(* Logix 5000 project; controller Reto1_SCADA Emulate 5570 rev 30.12; software revision 30.00 *)

TASK MainTask (continuous, watchdog 500 ms) : MainProgram

MODULES
   Local : Emulate 5570 (ICP 2, rev 30.12)
      I_O : vendor 1 type 0 code 15 (ICP 3, rev 1.1, Output RPI 150 ms)
END_MODULES

VAR_GLOBAL   (* controller tags *)
   Ambas : BOOL;
   Avanza_Exit : BOOL;
   BandaCorrecta : BOOL := 1;
   Bandera : BOOL := 1;
   BanderaA : BOOL;
   BanderaAmbas : BOOL;
   BanderaV : BOOL;
   BanExitA : BOOL;
   BanExiV : BOOL;
   BanSenA : BOOL;
   BanSenV : BOOL;
   ContadorA : COUNTER := (ACC := 10);
   ContadorV : COUNTER := (ACC := 10);
   Detener_Exit : BOOL;
   FIO_Avanzar : BOOL;
   FIO_AvanzarA : BOOL := 1;
   FIO_AvanzarUPA : BOOL := 1;
   FIO_AvanzarUPV : BOOL := 1;
   FIO_AvanzarV : BOOL := 1;
   FIO_Banda1 : BOOL := 1;
   FIO_Banda1b : BOOL := 1;
   FIO_Banda2 : BOOL := 1;
   FIO_Banda2b : BOOL := 1;
   FIO_BanderaBanda : BOOL;
   FIO_BanderaBandaA : BOOL;
   FIO_BanderaBandaV : BOOL;
   FIO_Detener : BOOL;
   FIO_DetenerA : BOOL;
   FIO_DetenerV : BOOL;
   FIO_Iniciar : BOOL;
   FIO_IniciarA : BOOL;
   FIO_IniciarV : BOOL;
   FIO_ParadaUPA : BOOL;
   FIO_ParadaUPV : BOOL;
   FIO_PusherAzul : BOOL;
   FIO_PusherVerde : BOOL;
   FIO_SensorAzul : BOOL;
   FIO_SensorExitA : BOOL;
   FIO_SensorExitV : BOOL;
   FIO_SensorPaso1 : BOOL;
   FIO_SensorPaso2 : BOOL;
   FIO_SensorVerde : BOOL;
   FIO_Start : BOOL;
   FIO_Stop : BOOL := 1;
   FIO_Stop_emergencia : BOOL := 1;
   FlancoBajadaA : BOOL;
   FlancoBajadaExA : BOOL;
   FlancoBajadaExV : BOOL;
   FlancoBajadaV : BOOL;
   TimerAvan : TIMER := (PRE := 1000, ACC := 25, EN := 1, TT := 1);
   TimerAvanV : TIMER := (PRE := 1000, ACC := 22, EN := 1, TT := 1);
   TimerBanda : TIMER := (PRE := 3000);
   TimerBandaV : TIMER := (PRE := 3000);
   TimerBien : TIMER := (PRE := 500, ACC := 510, EN := 1, DN := 1);
   TimerInicio : TIMER := (PRE := 2000, ACC := 2022, EN := 1, DN := 1);
   TimerInicioV : TIMER := (PRE := 2000, ACC := 2015, EN := 1, DN := 1);
   TimerP : TIMER := (PRE := 4000);
   TimerPUN : TIMER := (PRE := 3000, ACC := 2020, TT := 1, DN := 1);
   TimerPUNV : TIMER := (PRE := 3000, ACC := 2015, TT := 1, DN := 1);
   TimerPV : TIMER := (PRE := 4000);
   TimerStart : TIMER := (PRE := 4000);
END_VAR

PROGRAM MainProgram   (* main routine MainRoutine *)

ROUTINE Azul   (* ladder *)
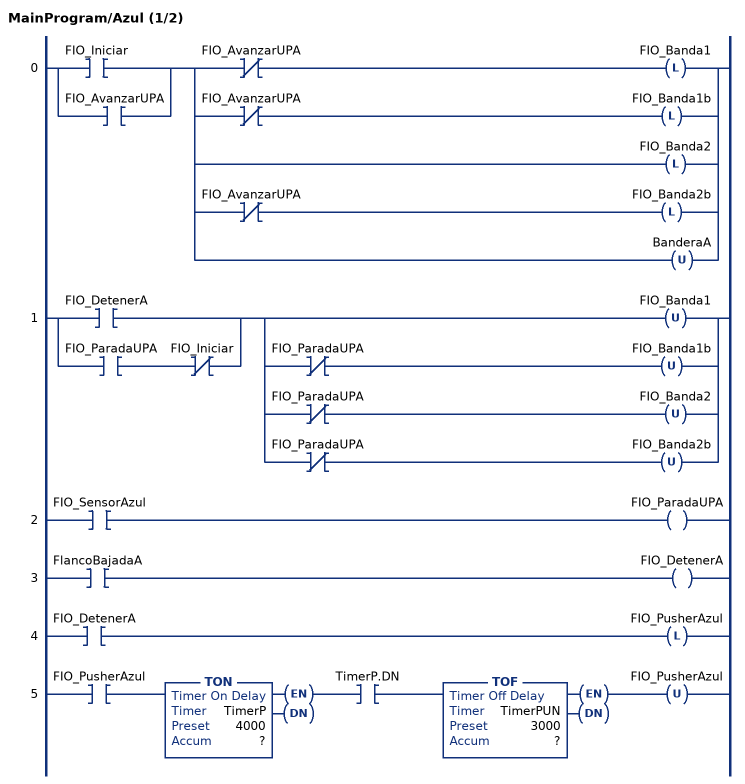
   0: [XIC(FIO_Iniciar) ,XIC(FIO_AvanzarUPA) ][XIO(FIO_AvanzarUPA) OTL(FIO_Banda1) ,XIO(FIO_AvanzarUPA) OTL(FIO_Banda1b) ,OTL(FIO_Banda2) ,XIO(FIO_AvanzarUPA) OTL(FIO_Banda2b) ,OTU(BanderaA) ];
   1: [XIC(FIO_DetenerA) ,XIC(FIO_ParadaUPA) XIO(FIO_Iniciar) ][OTU(FIO_Banda1) ,XIO(FIO_ParadaUPA) OTU(FIO_Banda1b) ,XIO(FIO_ParadaUPA) OTU(FIO_Banda2) ,XIO(FIO_ParadaUPA) OTU(FIO_Banda2b) ];
   2: XIC(FIO_SensorAzul)OTE(FIO_ParadaUPA);
   3: XIC(FlancoBajadaA)OTE(FIO_DetenerA);
   4: XIC(FIO_DetenerA)OTL(FIO_PusherAzul);
   5: XIC(FIO_PusherAzul)TON(TimerP,?,?)XIC(TimerP.DN)TOF(TimerPUN,?,?)OTU(FIO_PusherAzul);
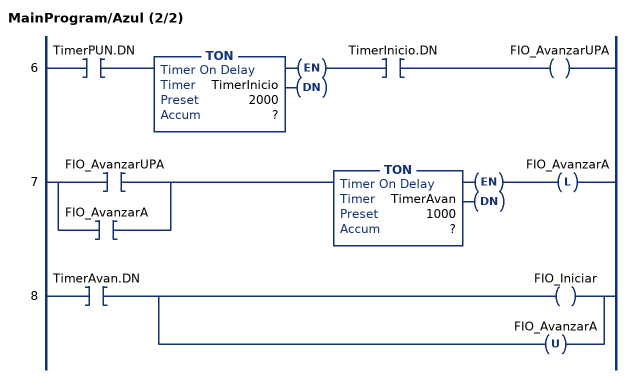
   6: XIC(TimerPUN.DN)TON(TimerInicio,?,?)XIC(TimerInicio.DN)OTE(FIO_AvanzarUPA);
   7: [XIC(FIO_AvanzarUPA) ,XIC(FIO_AvanzarA) ]TON(TimerAvan,?,?)OTL(FIO_AvanzarA);
   8: XIC(TimerAvan.DN)[OTE(FIO_Iniciar) ,OTU(FIO_AvanzarA) ];
END_ROUTINE

ROUTINE MainRoutine   (* ladder *)
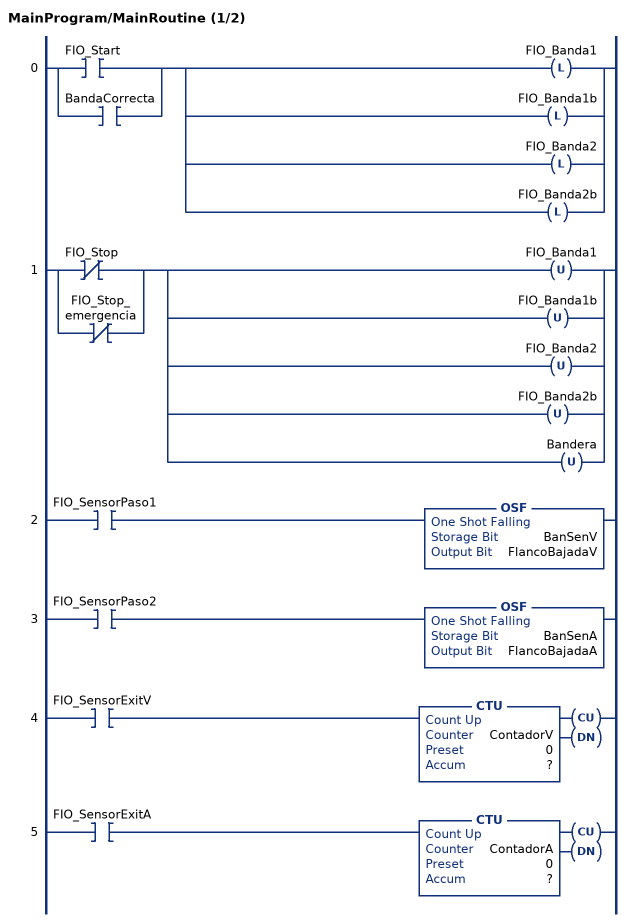
   0: [XIC(FIO_Start) ,XIC(BandaCorrecta) ][OTL(FIO_Banda1) ,OTL(FIO_Banda1b) ,OTL(FIO_Banda2) ,OTL(FIO_Banda2b) ];
   1: [XIO(FIO_Stop) ,XIO(FIO_Stop_emergencia) ][OTU(FIO_Banda1) ,OTU(FIO_Banda1b) ,OTU(FIO_Banda2) ,OTU(FIO_Banda2b) ,OTU(Bandera) ];
   2: XIC(FIO_SensorPaso1)OSF(BanSenV,FlancoBajadaV);
   3: XIC(FIO_SensorPaso2)OSF(BanSenA,FlancoBajadaA);
   4: XIC(FIO_SensorExitV)CTU(ContadorV,?,?);
   5: XIC(FIO_SensorExitA)CTU(ContadorA,?,?);
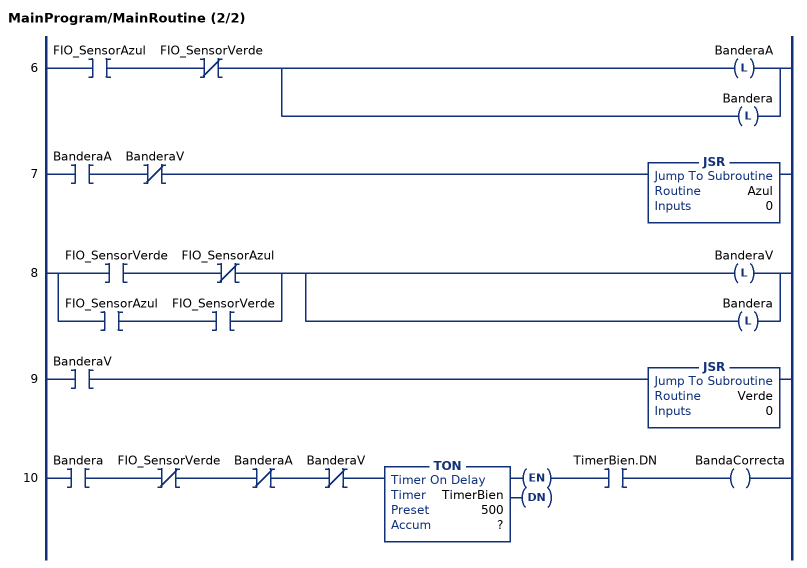
   6: XIC(FIO_SensorAzul)XIO(FIO_SensorVerde)[OTL(BanderaA) ,OTL(Bandera) ];
   7: XIC(BanderaA)XIO(BanderaV)JSR(Azul,0);
   8: [XIC(FIO_SensorVerde) XIO(FIO_SensorAzul) ,XIC(FIO_SensorAzul) XIC(FIO_SensorVerde) ][OTL(BanderaV) ,OTL(Bandera) ];
   9: XIC(BanderaV)JSR(Verde,0);
   10: XIC(Bandera)XIO(FIO_SensorVerde)XIO(BanderaA)XIO(BanderaV)TON(TimerBien,?,?)XIC(TimerBien.DN)OTE(BandaCorrecta);
END_ROUTINE

ROUTINE Verde   (* ladder *)
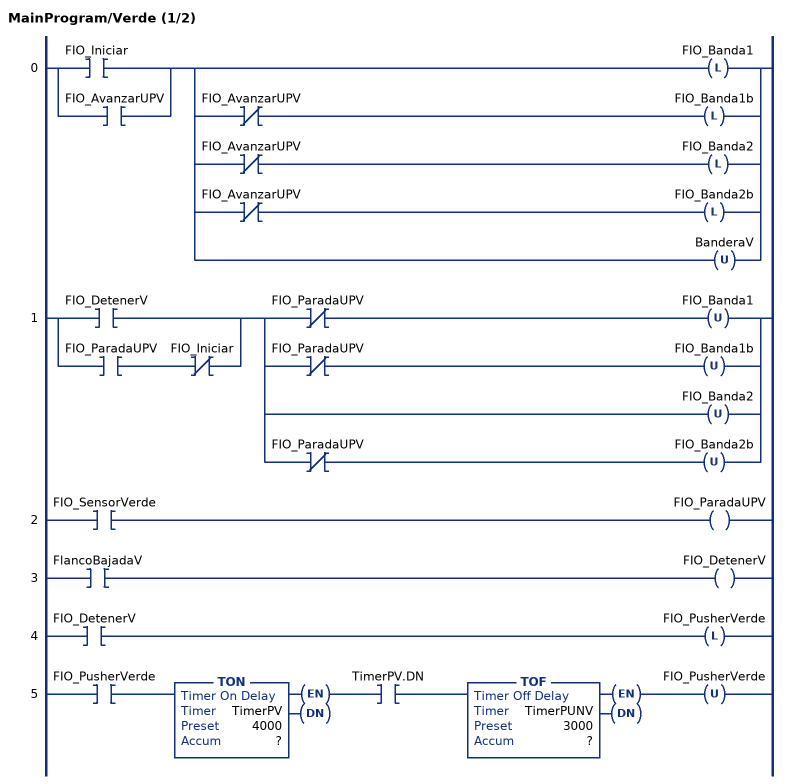
   0: [XIC(FIO_Iniciar) ,XIC(FIO_AvanzarUPV) ][OTL(FIO_Banda1) ,XIO(FIO_AvanzarUPV) OTL(FIO_Banda1b) ,XIO(FIO_AvanzarUPV) OTL(FIO_Banda2) ,XIO(FIO_AvanzarUPV) OTL(FIO_Banda2b) ,OTU(BanderaV) ];
   1: [XIC(FIO_DetenerV) ,XIC(FIO_ParadaUPV) XIO(FIO_Iniciar) ][XIO(FIO_ParadaUPV) OTU(FIO_Banda1) ,XIO(FIO_ParadaUPV) OTU(FIO_Banda1b) ,OTU(FIO_Banda2) ,XIO(FIO_ParadaUPV) OTU(FIO_Banda2b) ];
   2: XIC(FIO_SensorVerde)OTE(FIO_ParadaUPV);
   3: XIC(FlancoBajadaV)OTE(FIO_DetenerV);
   4: XIC(FIO_DetenerV)OTL(FIO_PusherVerde);
   5: XIC(FIO_PusherVerde)TON(TimerPV,?,?)XIC(TimerPV.DN)TOF(TimerPUNV,?,?)OTU(FIO_PusherVerde);
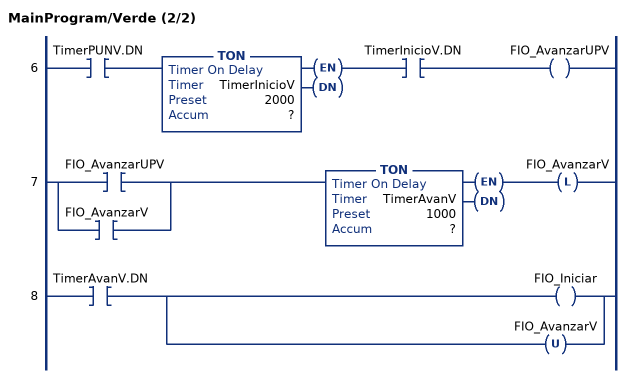
   6: XIC(TimerPUNV.DN)TON(TimerInicioV,?,?)XIC(TimerInicioV.DN)OTE(FIO_AvanzarUPV);
   7: [XIC(FIO_AvanzarUPV) ,XIC(FIO_AvanzarV) ]TON(TimerAvanV,?,?)OTL(FIO_AvanzarV);
   8: XIC(TimerAvanV.DN)[OTE(FIO_Iniciar) ,OTU(FIO_AvanzarV) ];
END_ROUTINE
END_PROGRAM
